FUNCTION F_RaiseAlarmWithStringParameters : BOOL
VAR_IN_OUT
    fbAlarm : FB_TcAlarm; //Alarm to be raised
END_VAR
VAR_INPUT
    sString_1 : STRING;
    sString_2 : STRING;
    sString_3 : STRING;
END_VAR

fbAlarm.ipArguments.Clear();

IF sString_1 <> '' THEN
    fbAlarm.ipArguments.AddString(sString_1);
END_IF

IF sString_2 <> '' THEN
    fbAlarm.ipArguments.AddString(sString_2);
END_IF

IF sString_3 <> '' THEN
    fbAlarm.ipArguments.AddString(sString_3);
END_IF

fbAlarm.Raise(0);

END_FUNCTION

(* stored: Version 1.1.0.1, ProductVersion 3.1.4024.11
   POU F_RaiseAlarmWithStringParameters: Id {0fae160d-14c3-4278-8cd1-635da75444f7}, SpecialFunc None *)
